// TIA Portal project "PLCII_Pro8" (V15.1)

(* hardware
DEVICE "S7-1200 station_1"  S7-1200 Station
   slot 0: "Rack_0"  S7-1200 Rack  Rack  V1.0
   slot 1: "PLC_1"  CPU 1215C DC/DC/Rly  6ES7 215-1HG40-0XB0  V4.2
*)

// ===== PLC "PLC_1"  CPU 1215C DC/DC/Rly =====

VAR_GLOBAL   // PLC tag table "Default tag table"
   "Start" AT %M0.0 : Bool;
   "Sys_runing" AT %M0.1 : Bool;
   "Stop" AT %M0.2 : Bool;
   "Activate" AT %M0.3 : Bool;
   "Sys_Activated" AT %M0.4 : Bool;
END_VAR

DATA_BLOCK "SysVaribales"   // DB1
{ S7_Optimized_Access := 'TRUE' }
VERSION : 0.1
   VAR
      PumpSpeed : Int;
      PumpDirection : Int;
      Sp_vacuum : Int;
      AC_vacuum : Int;
      MeasuredValue : Int;
      State_OF_measurment : String;
      PumpRuningSpeed : Int;
   END_VAR
BEGIN
END_DATA_BLOCK

DATA_BLOCK "VFD_Control_DB"   // DB2
{ S7_Optimized_Access := 'TRUE' }
VERSION : 0.1
// stored: InstanceOfName VFD_Control
"VFD_Control"
BEGIN
END_DATA_BLOCK

FUNCTION_BLOCK "VFD_Control"   // FB1, LAD
{ S7_Optimized_Access := 'TRUE' }
VERSION : 0.1
   VAR_INPUT
      Excute : Bool;
      Sp_vacuum : Int;
      Time_BW_Read : Time;
   END_VAR
   VAR_IN_OUT
      AC_vacuum : Int;
   END_VAR
   VAR
      IEC_Timer_0_Instance : TON_TIME;
      ons1 : Bool;
      ons2 : Bool;
      ons3 : Bool;
      ons4 : Bool;
      ons5 : Bool;
      ons6 : Bool;
      ons7 : Bool;
      ons8 : Bool;
      ons9 : Bool;
      ons10 : Bool;
      Used_vacuum : Int;
      varp : Int;
   END_VAR
   VAR_TEMP
      AC_vacuum_Normalized : Real;
      AC_vacuum_Scaled : Int;
   END_VAR
BEGIN

REGION Network 1
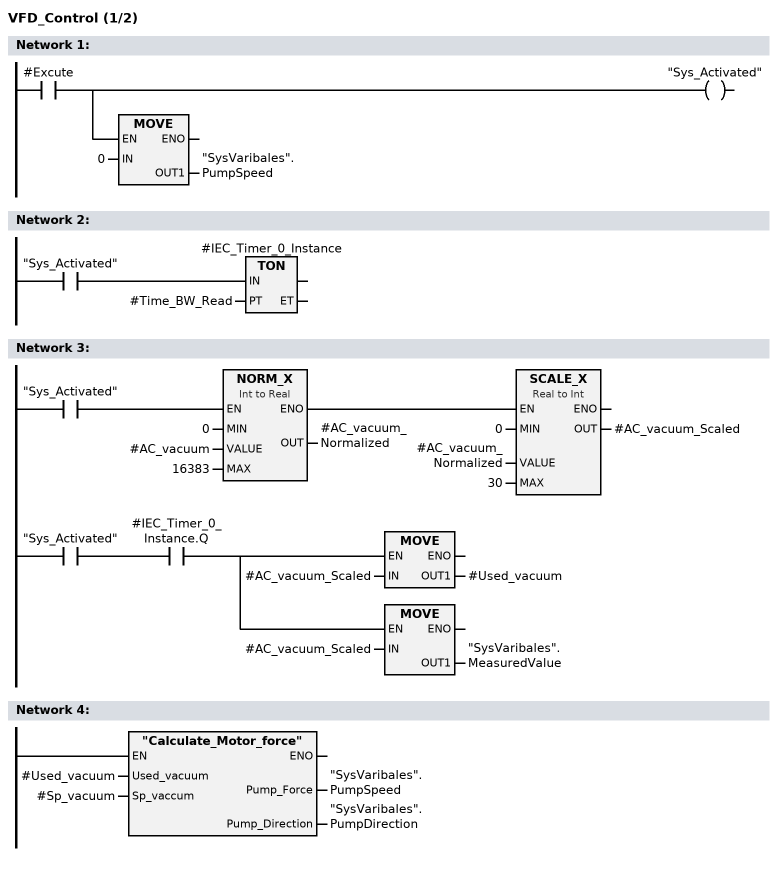
   RUNG wire#powerrail
      Contact( #Excute )
      wire#w1
      Coil( "Sys_Activated" )
   END_RUNG
   RUNG wire#w1
      Move(in := 0, out1 => "SysVaribales".PumpSpeed)
   END_RUNG
   // the same network as SCL:
   "Sys_Activated" := #Excute;
   IF #Excute THEN "SysVaribales".PumpSpeed := 0; END_IF;
END_REGION

REGION Network 2
   #IEC_Timer_0_Instance(IN := "Sys_Activated", PT := #Time_BW_Read);   // TON
END_REGION

REGION Network 3
   RUNG wire#powerrail
      Contact( "Sys_Activated" )
      { S7_Templates := "[SrcType := Int, DestType := Real]" } Normalize(min := 0, value := #AC_vacuum, max := 16383, out => #AC_vacuum_Normalized)
      { S7_Templates := "[SrcType := Real, DestType := Int]" } Scale(min := 0, value := #AC_vacuum_Normalized, max := 30, out => #AC_vacuum_Scaled)
   END_RUNG
   RUNG wire#powerrail
      Contact( "Sys_Activated" )
      Contact( #IEC_Timer_0_Instance.Q )
      wire#w1
      Move(in := #AC_vacuum_Scaled, out1 => #Used_vacuum)
   END_RUNG
   RUNG wire#w1
      Move(in := #AC_vacuum_Scaled, out1 => "SysVaribales".MeasuredValue)
   END_RUNG
   // the same network as SCL:
   IF "Sys_Activated" THEN
       #AC_vacuum_Normalized := NORM_X(MIN := 0, VALUE := #AC_vacuum, MAX := 16383);
       #AC_vacuum_Scaled := SCALE_X(MIN := 0, VALUE := #AC_vacuum_Normalized, MAX := 30);
   END_IF;
   IF "Sys_Activated" AND #IEC_Timer_0_Instance.Q THEN
       #Used_vacuum := #AC_vacuum_Scaled;
       "SysVaribales".MeasuredValue := #AC_vacuum_Scaled;
   END_IF;
END_REGION

REGION Network 4
   RUNG wire#powerrail
      "Calculate_Motor_force"(Used_vacuum := #Used_vacuum, Sp_vaccum := #Sp_vacuum, Pump_Force => "SysVaribales".PumpSpeed, Pump_Direction => "SysVaribales".PumpDirection)
   END_RUNG
   // the same network as SCL:
   "Calculate_Motor_force"(Used_vacuum := #Used_vacuum,
                           Sp_vaccum := #Sp_vacuum,
                           Pump_Force => "SysVaribales".PumpSpeed,
                           Pump_Direction => "SysVaribales".PumpDirection);
END_REGION

REGION Network 5
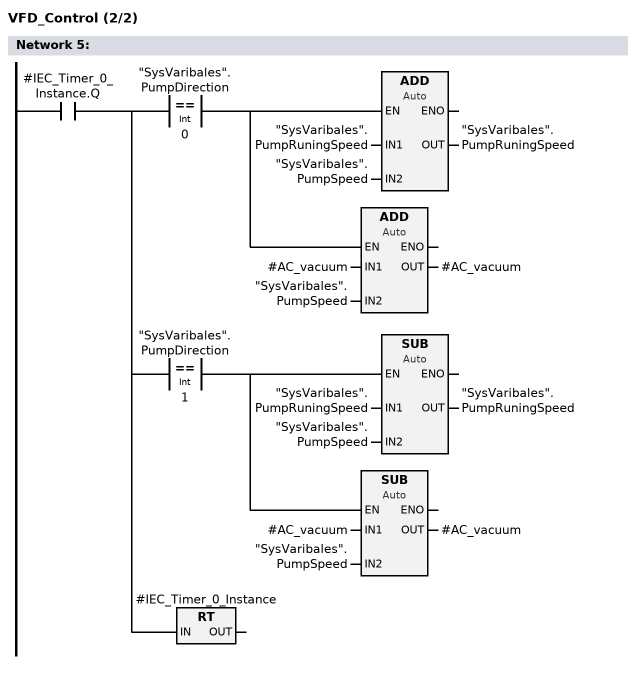
   RUNG wire#powerrail
      Contact( #IEC_Timer_0_Instance.Q )
      wire#w1
      { S7_Templates := "SrcType := Int" } EQ_Contact(in1 := "SysVaribales".PumpDirection, in2 := 0)
      wire#w2
      Add(in1 := "SysVaribales".PumpRuningSpeed, in2 := "SysVaribales".PumpSpeed, out => "SysVaribales".PumpRuningSpeed)
   END_RUNG
   RUNG wire#w2
      Add(in1 := #AC_vacuum, in2 := "SysVaribales".PumpSpeed, out => #AC_vacuum)
   END_RUNG
   RUNG wire#w1
      { S7_Templates := "SrcType := Int" } EQ_Contact(in1 := "SysVaribales".PumpDirection, in2 := 1)
      wire#w3
      Sub(in1 := "SysVaribales".PumpRuningSpeed, in2 := "SysVaribales".PumpSpeed, out => "SysVaribales".PumpRuningSpeed)
   END_RUNG
   RUNG wire#w3
      Sub(in1 := #AC_vacuum, in2 := "SysVaribales".PumpSpeed, out => #AC_vacuum)
   END_RUNG
   RUNG wire#w1
      RT_Coil( #IEC_Timer_0_Instance )
   END_RUNG
   // the same network as SCL:
   IF #IEC_Timer_0_Instance.Q AND ("SysVaribales".PumpDirection = 0) THEN
       "SysVaribales".PumpRuningSpeed := "SysVaribales".PumpRuningSpeed + "SysVaribales".PumpSpeed;
       #AC_vacuum := #AC_vacuum + "SysVaribales".PumpSpeed;
   END_IF;
   IF #IEC_Timer_0_Instance.Q AND ("SysVaribales".PumpDirection = 1) THEN
       "SysVaribales".PumpRuningSpeed := "SysVaribales".PumpRuningSpeed - "SysVaribales".PumpSpeed;
       #AC_vacuum := #AC_vacuum - "SysVaribales".PumpSpeed;
   END_IF;
   IF #IEC_Timer_0_Instance.Q THEN RESET_TIMER(#IEC_Timer_0_Instance); END_IF;
END_REGION
END_FUNCTION_BLOCK

FUNCTION "Calculate_Motor_force" : Void   // FC1, LAD
{ S7_Optimized_Access := 'TRUE' }
VERSION : 0.1
   VAR_INPUT
      Used_vacuum : Int;
      Sp_vaccum : Int;
   END_VAR
   VAR_OUTPUT
      Pump_Force : Int;
      Pump_Direction : Int;
   END_VAR
   VAR_TEMP
      Used_Diff_vacuum_temp : Real;
      Used_Diff_vacuum_temp_1 : Real;
   END_VAR
BEGIN

REGION Network 1: GettingValues
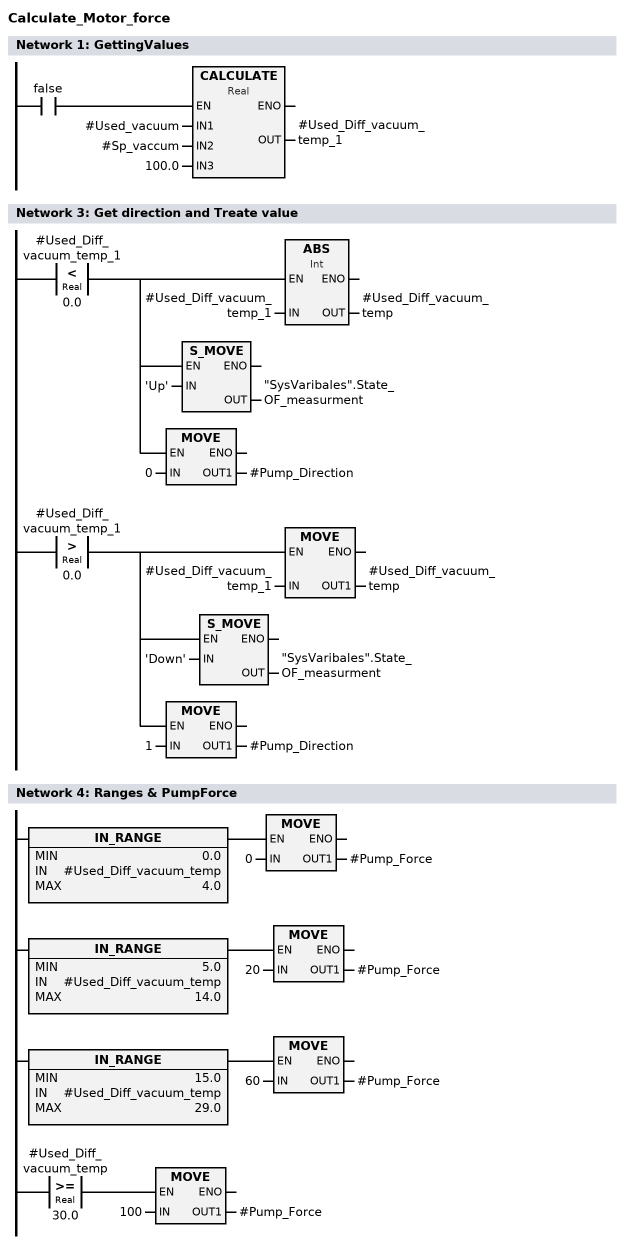
   RUNG wire#powerrail
      Contact( false )
      { S7_Templates := "SrcType := Real"; S7_Expression := "((IN1-IN2)/IN2)* IN3" } Calculate(in1 := #Used_vacuum, in2 := #Sp_vaccum, in3 := 100.0, out => #Used_Diff_vacuum_temp_1)
   END_RUNG
   // the same network as SCL:
   IF false THEN #Used_Diff_vacuum_temp_1 := ((#Used_vacuum-#Sp_vaccum)/#Sp_vaccum)* 100.0; END_IF;
END_REGION

REGION Network 2 (SCL)
   #Used_Diff_vacuum_temp_1 := ((INT_TO_REAL(#Used_vacuum) - INT_TO_REAL(#Sp_vaccum))/#Sp_vaccum) *100 ;
END_REGION

REGION Network 3: Get direction and Treate value
   RUNG wire#powerrail
      { S7_Templates := "SrcType := Real" } LT_Contact(in1 := #Used_Diff_vacuum_temp_1, in2 := 0.0)
      wire#w1
      { S7_Templates := "SrcType := Int" } Abs(in := #Used_Diff_vacuum_temp_1, out => #Used_Diff_vacuum_temp)
   END_RUNG
   RUNG wire#w1
      S_Move(in := 'Up', out => "SysVaribales".State_OF_measurment)
   END_RUNG
   RUNG wire#w1
      Move(in := 0, out1 => #Pump_Direction)
   END_RUNG
   RUNG wire#powerrail
      { S7_Templates := "SrcType := Real" } GT_Contact(in1 := #Used_Diff_vacuum_temp_1, in2 := 0.0)
      wire#w2
      Move(in := #Used_Diff_vacuum_temp_1, out1 => #Used_Diff_vacuum_temp)
   END_RUNG
   RUNG wire#w2
      S_Move(in := 'Down', out => "SysVaribales".State_OF_measurment)
   END_RUNG
   RUNG wire#w2
      Move(in := 1, out1 => #Pump_Direction)
   END_RUNG
   // the same network as SCL:
   IF #Used_Diff_vacuum_temp_1 < 0.0 THEN
       #Used_Diff_vacuum_temp := ABS(#Used_Diff_vacuum_temp_1);
       "SysVaribales".State_OF_measurment := 'Up';
       #Pump_Direction := 0;
   END_IF;
   IF #Used_Diff_vacuum_temp_1 > 0.0 THEN
       #Used_Diff_vacuum_temp := #Used_Diff_vacuum_temp_1;
       "SysVaribales".State_OF_measurment := 'Down';
       #Pump_Direction := 1;
   END_IF;
END_REGION

REGION Network 4: Ranges & PumpForce
   RUNG wire#powerrail
      { S7_Templates := "SrcType := Real" } InRange(min := 0.0, in := #Used_Diff_vacuum_temp, max := 4.0)
      Move(in := 0, out1 => #Pump_Force)
   END_RUNG
   RUNG wire#powerrail
      { S7_Templates := "SrcType := Real" } InRange(min := 5.0, in := #Used_Diff_vacuum_temp, max := 14.0)
      Move(in := 20, out1 => #Pump_Force)
   END_RUNG
   RUNG wire#powerrail
      { S7_Templates := "SrcType := Real" } InRange(min := 15.0, in := #Used_Diff_vacuum_temp, max := 29.0)
      Move(in := 60, out1 => #Pump_Force)
   END_RUNG
   RUNG wire#powerrail
      { S7_Templates := "SrcType := Real" } GE_Contact(in1 := #Used_Diff_vacuum_temp, in2 := 30.0)
      Move(in := 100, out1 => #Pump_Force)
   END_RUNG
   // the same network as SCL:
   IF (0.0 <= #Used_Diff_vacuum_temp) AND (#Used_Diff_vacuum_temp <= 4.0) THEN #Pump_Force := 0; END_IF;
   IF (5.0 <= #Used_Diff_vacuum_temp) AND (#Used_Diff_vacuum_temp <= 14.0) THEN #Pump_Force := 20; END_IF;
   IF (15.0 <= #Used_Diff_vacuum_temp) AND (#Used_Diff_vacuum_temp <= 29.0) THEN #Pump_Force := 60; END_IF;
   IF #Used_Diff_vacuum_temp >= 30.0 THEN #Pump_Force := 100; END_IF;
END_REGION
END_FUNCTION

ORGANIZATION_BLOCK "Main"   // OB1, LAD, ProgramCycle
TITLE = "Main Program Sweep (Cycle)"
{ S7_Optimized_Access := 'TRUE' }
VERSION : 0.1
   VAR_INPUT
      Initial_Call : Bool;   // Initial call of this OB
      Remanence : Bool;   // =True, if remanent data are available
   END_VAR
BEGIN

REGION Network 1
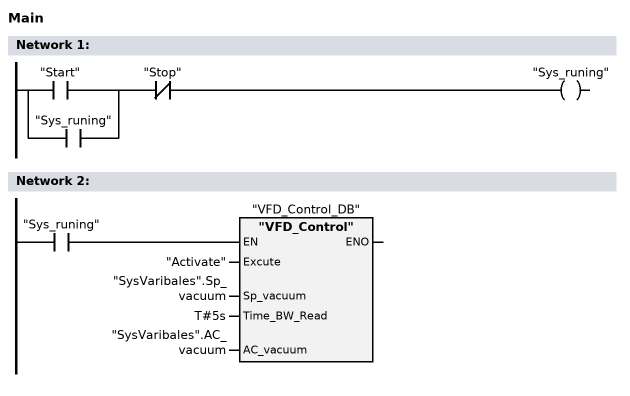
   RUNG wire#powerrail
      Contact( "Start" )
      wire#w1
      I_Contact( "Stop" )
      Coil( "Sys_runing" )
   END_RUNG
   RUNG wire#powerrail
      Contact( "Sys_runing" )
   END_RUNG wire#w1
   // the same network as SCL:
   "Sys_runing" := ("Start" OR "Sys_runing") AND NOT "Stop";
END_REGION

REGION Network 2
   RUNG wire#powerrail
      Contact( "Sys_runing" )
      "VFD_Control_DB"(Excute := "Activate", Sp_vacuum := "SysVaribales".Sp_vacuum, Time_BW_Read := T#5s, AC_vacuum := "SysVaribales".AC_vacuum)
   END_RUNG
   // the same network as SCL:
   IF "Sys_runing" THEN
       "VFD_Control_DB"(Excute := "Activate",   // "VFD_Control"
                        Sp_vacuum := "SysVaribales".Sp_vacuum,
                        Time_BW_Read := T#5s,
                        AC_vacuum := "SysVaribales".AC_vacuum);
   END_IF;
END_REGION
END_ORGANIZATION_BLOCK